SUBAPPLICATION Uebung_015 (* Object Pointer umschalten *)
  (* Standard: 61499-2; Description: Copyright (c) 2023 Meisterschulen am Ostbahnhof This program and the accompanying materials are made available under the terms of the Eclipse Public License 2.0 which is available at https://www.eclipse.org/legal/epl-2.0/ SPDX-License-Identifier: EPL-2.0 *)
  (* Version 1.0, 2023-10-23, Franz Höpfinger, Meisterschulen am Ostbahnhof, initial API and implementation and/or initial documentation *)
  PACKAGE Uebungen;
  IMPORT isobus::UT::io::Softkey::SoftKeyActivationCode::SK_RELEASED;
  IMPORT Uebungen::const::UT::DefaultPool::Button_A1;
  IMPORT Uebungen::const::UT::DefaultPool::ObjectPointer_P1;
  IMPORT Uebungen::const::UT::DefaultPool::SoftKey_F1;
  IMPORT Uebungen::const::UT::DefaultPool::SoftKey_F2;
  IMPORT isobus::UT::Q::const::IDs::ID_NULL;
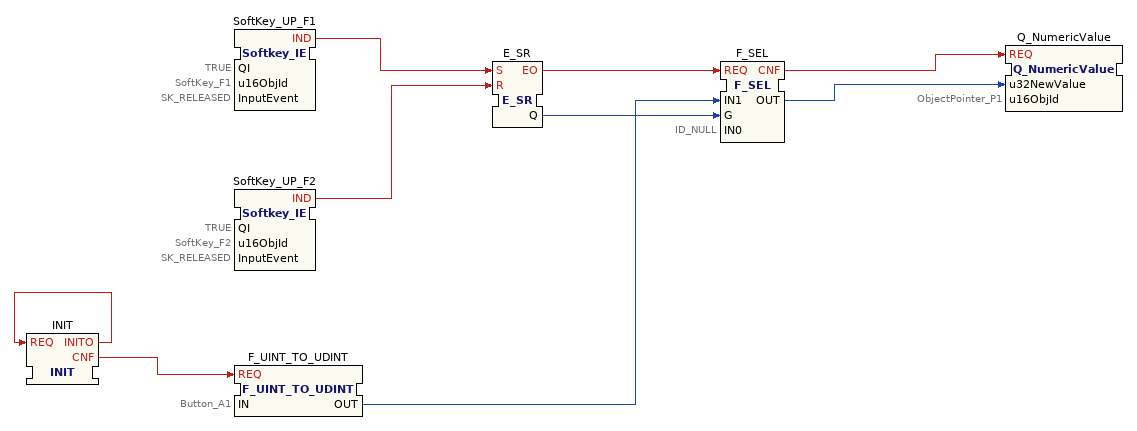
  FBS
    SoftKey_UP_F1 : isobus::UT::io::Softkey::Softkey_IE(QI := TRUE, u16ObjId := SoftKey_F1, InputEvent := SK_RELEASED);
    SoftKey_UP_F2 : isobus::UT::io::Softkey::Softkey_IE(QI := TRUE, u16ObjId := SoftKey_F2, InputEvent := SK_RELEASED);
    E_SR : iec61499::events::E_SR;
    F_UINT_TO_UDINT : iec61131::conversion::F_UINT_TO_UDINT(IN := Button_A1);
    F_SEL : iec61131::selection::F_SEL(IN0 := ID_NULL);
    Q_NumericValue : isobus::UT::Q::Q_NumericValue(u16ObjId := ObjectPointer_P1);
    INIT : iec61131::booleanOperators::INIT;
  END_FBS
  EVENT_CONNECTIONS
    SoftKey_UP_F1.IND TO E_SR.S;
    SoftKey_UP_F2.IND TO E_SR.R;
    F_SEL.CNF TO Q_NumericValue.REQ;
    E_SR.EO TO F_SEL.REQ;
    INIT.INITO TO INIT.REQ;
    INIT.CNF TO F_UINT_TO_UDINT.REQ;
  END_CONNECTIONS
  DATA_CONNECTIONS
    F_SEL.OUT TO Q_NumericValue.u32NewValue;
    F_UINT_TO_UDINT.OUT TO F_SEL.IN1;
    E_SR.Q TO F_SEL.G;
  END_CONNECTIONS
END_SUBAPPLICATION
